Fanuc KAREL source: kt00334.KL

-- PROVISIONAL review KL for V770-1; original PC SHA256 8c1f47721bb6027ca8de52be89abc352f8972bad77ebe535064a5fcf860bc259
-- Incomplete behavior may be omitted. Consult companion uncertainty JSON. Do not deploy.
PROGRAM KT00334
%NOLOCKGROUP
VAR
  R1 : REAL
  R2 : REAL
  OUT : BOOLEAN
BEGIN
  -- UNRESOLVED_PC offsets 5-16; opcodes 2E,23
  -- UNRESOLVED_PC offsets 21-32; opcodes 2E,23
  -- UNRESOLVED_PC offsets 37-48; opcodes 2E,23
  -- UNRESOLVED_PC offsets 53-64; opcodes 2E,23
  -- UNRESOLVED_PC offsets 69-88; opcodes 21,21,6F,23
  -- UNRESOLVED_PC offsets 93-97; opcodes 7F
END KT00334
